// TIA Portal project "three_head" (V16)

(* hardware
DEVICE "S71500/ET200MP station_1"  S7-1500 station
   slot 0: "Rail_0"  Rack  6ES7 590-1***0-0AA0
   slot 1: "PLC_1"  CPU 1512C-1 PN  6ES7 512-1CK00-0AB0  V1.8
      slot 3: "CPU display_1"  6ES7591-1AA00-0AA0
      slot 32768: "PROFINET interface_1"  X1
         slot 32769: "Port_1"  X1 P1
         slot 32770: "Port_2"  X1 P2
*)

// ===== PLC "PLC_1"  CPU 1512C-1 PN =====

VAR_GLOBAL   // PLC tag table "Default tag table"
   "L-1" AT %IW0 : Int;   // level tank indicator, 0-100 L
   "K-1" AT %I10.0 : Bool;   // agitator
   "liter" AT %IW4 : Int;
   "Clock_Byte" AT %MB0 : Byte;
   "Clock_10Hz" AT %M0.0 : Bool;
   "Clock_5Hz" AT %M0.1 : Bool;
   "Clock_2.5Hz" AT %M0.2 : Bool;
   "Clock_2Hz" AT %M0.3 : Bool;
   "Clock_1.25Hz" AT %M0.4 : Bool;
   "Clock_1Hz" AT %M0.5 : Bool;
   "Clock_0.625Hz" AT %M0.6 : Bool;
   "Clock_0.5Hz" AT %M0.7 : Bool;
   "on button" AT %M1.0 : Bool;
END_VAR

DATA_BLOCK "Block_1_DB"   // DB2
{ S7_Optimized_Access := 'TRUE' }
VERSION : 0.1
// stored: InstanceOfName FB to valve control
"FB to valve control"
BEGIN
END_DATA_BLOCK

// folder: System blocks/Program resources

DATA_BLOCK "IEC_Timer_0_DB"   // DB1
{ S7_Optimized_Access := 'TRUE' }
AUTHOR : Simatic
FAMILY : IEC
NAME : IEC_TMR
VERSION : 1.0
// stored: InstanceOfName IEC_TIMER
"IEC_TIMER"
BEGIN
END_DATA_BLOCK

// folder: (top level)

FUNCTION_BLOCK "FB to valve control"   // FB1, SCL
{ S7_Optimized_Access := 'TRUE' }
VERSION : 0.1
   VAR_INPUT
      liq_level : Real;
   END_VAR
   VAR_OUTPUT
      agitator : Bool;
   END_VAR
   VAR CONSTANT
      desirable_liq_level : Real := 30.0;
   END_VAR
BEGIN
   #liq_level := 0.0; // Correct, cause assignment with
   //default value of data type 0.0
   // Correct --> Working with constants
   IF (ABS(#liq_level) = #desirable_liq_level) THEN
       #agitator := TRUE;
   ELSE
       #agitator := FALSE;
   END_IF;
END_FUNCTION_BLOCK

FUNCTION "rawdata to liter" : Void   // FC2, LAD
{ S7_Optimized_Access := 'TRUE' }
VERSION : 0.1
   VAR_INPUT
      rawinput : Int;
   END_VAR
   VAR_OUTPUT
      liter : Real;
   END_VAR
   VAR_TEMP
      percent : Real;
   END_VAR
BEGIN

REGION Network 1
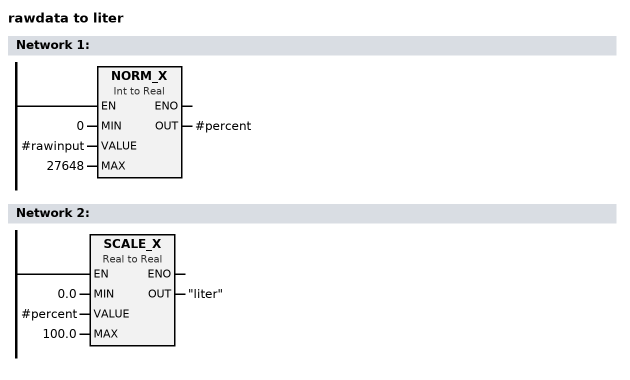
   RUNG wire#powerrail
      { S7_Templates := "[SrcType := Int, DestType := Real]" } Normalize(min := 0, value := #rawinput, max := 27648, out => #percent)
   END_RUNG
   // the same network as SCL:
   #percent := NORM_X(MIN := 0, VALUE := #rawinput, MAX := 27648);
END_REGION

REGION Network 2
   RUNG wire#powerrail
      { S7_Templates := "[SrcType := Real, DestType := Real]" } Scale(min := 0.0, value := #percent, max := 100.0, out => "liter")
   END_RUNG
   // the same network as SCL:
   "liter" := SCALE_X(MIN := 0.0, VALUE := #percent, MAX := 100.0);
END_REGION
END_FUNCTION

ORGANIZATION_BLOCK "Main"   // OB1, LAD, ProgramCycle
TITLE = "Main Program Sweep (Cycle)"
{ S7_Optimized_Access := 'TRUE' }
VERSION : 0.1
   VAR_INPUT
      Initial_Call : Bool;   // Initial call of this OB
      Remanence : Bool;   // =True, if remanent data are available
   END_VAR
BEGIN

REGION Network 1
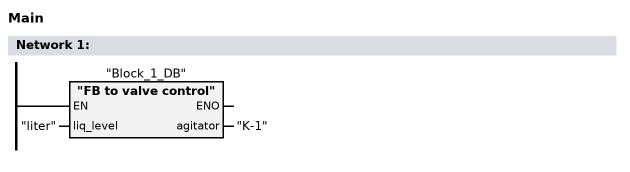
   RUNG wire#powerrail
      "Block_1_DB"(liq_level := "liter", agitator => "K-1")
   END_RUNG
   // the same network as SCL:
   "Block_1_DB"(liq_level := "liter", agitator => "K-1");   // "FB to valve control"
END_REGION
END_ORGANIZATION_BLOCK

ORGANIZATION_BLOCK "3_cycle update"   // OB123, LAD, ProgramCycle
TITLE = "Main Program Sweep (Cycle)"
{ S7_Optimized_Access := 'TRUE' }
VERSION : 0.1
   VAR_INPUT
      Initial_Call : Bool;   // Initial call of this OB
      Remanence : Bool;   // =True, if remanent data are available
   END_VAR
BEGIN

REGION Network 1
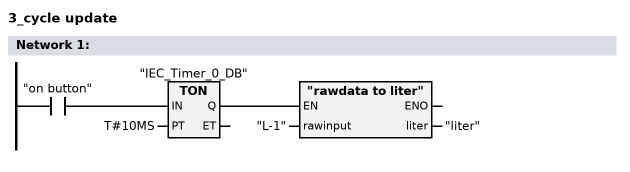
   "IEC_Timer_0_DB".TON(IN := "on button", PT := T#10MS);
   IF "IEC_Timer_0_DB".Q THEN "rawdata to liter"(rawinput := "L-1", liter => "liter"); END_IF;
END_REGION
END_ORGANIZATION_BLOCK